// TIA Portal V20 export
TYPE "typeCmControlNodeBrakeTest"
// stored: Namespace Unit1.Em6
   STRUCT
      visionUnit { ExternalWritable := 'False'} : "LER_typeBrakeTestEmControlNodes";
   END_STRUCT;
END_TYPE
